// TIA Portal V20 export
// export: Created 2025-12-01T14:56:19.1888575Z, ExportSetting None, DisplayName Totally Integrated Automation Portal, DisplayVersion V20 Update 3, DisplayName TIA Portal Openness, DisplayVersion V20 Update 3, DisplayName TIA Portal Version Control Interface, DisplayVersion V20 Update 3, DisplayName STEP 7 Professional, DisplayVersion V20 Update 3, DisplayName STEP 7 Safety, DisplayVersion V20 Update 2, DisplayName WinCC Basic/Comfort/Advanced, DisplayVersion V20 Update 3, DisplayName WinCC Professional, DisplayVersion V20 Update 3, DisplayName WinCC Unified, DisplayVersion V20 Update 3
TYPE "i550 Lenze_AS-i"
   STRUCT
      "Estatus variador (Inputs)" : Struct   // Word que informa del estado del dispositivo
         "Ready for operation" : Bool;
         "Auto setp active" : Bool;
         "Actual speed = 0" : Bool;
         "Fault active" : Bool;
         "Inverter disable" : Bool;
         "Current limit reached" : Bool;
         "Torque limit reached" : Bool;
         "Setpoint speed reached" : Bool;
         "Digital input 1" : Bool;
         "Digital input 2" : Bool;
         "Digital input 3" : Bool;
         "Digital input 4" : Bool;
         "Digital input 5" : Bool;
         Running : Bool;
         "Reserva 1" : Bool;
         "Reserva 2" : Bool;
      END_STRUCT;
      "Código de error (Inputs)" : UInt;   // Código proporcionado por Lenze para diagnosticar el fallo
      "Corriente actual (Inputs)" : UInt;   // Corriente actual en dispositivo. Formato 21 = 2,1 A
      "Palabra de control (Outputs)" : Struct   // Word que controla la activación del dispositvo
         "Run forward" : Bool;
         "Reverse rotation dirtect." : Bool;
         "Reset error" : Bool;
         "Position counter reset" : Bool;
         "Activate quick stop" : Bool;
         "Sel. paramset b0" : Bool;
         "Sel. paramset b1" : Bool;
         "Reserva 0.7" : Bool;
         "Reserva 1.0" : Bool;
         "Reserva 1.1" : Bool;
         "Reserva 1.2" : Bool;
         "Reserva 1.3" : Bool;
         "Reserva 1.4" : Bool;
         "Reserva 1.5" : Bool;
         "Reserva 1.6" : Bool;
         "Activar salida DO1" : Bool;
      END_STRUCT;
      "Consigna de frecuencia (Outputs)" : UInt;   // Frecuencia enviada al dispositivo. Formato 3250 = 32,50 Hz
      "ACC (Outputs)" : UInt := 10;   // 5->0,5sg; 10->1sg; 50->5sg; 100->10sg a Frecuencia máxima
      "DCC (Outputs)" : UInt := 10;   // 5->0,5sg; 10->1sg; 50->5sg; 100->10sg a Frecuencia máxima
      Direccion_Inicial_Nodo : Int;
      "Error activo" : Bool;
   END_STRUCT;
END_TYPE
